TYPE T_Whitespace_Location : E_WHITESPACE_LOCATION; END_TYPE

(* stored: Version 1.1.0.1, ProductVersion 3.1.4024.4
   DUT T_Whitespace_Location: Id {5081585d-551a-41ed-9fd2-e5c015a747af} *)
